{attribute 'pack_mode':='1'}
TYPE InitToteRequestParams :
STRUCT
	source_id : ModelIdentifier;
	target_id: ModelIdentifier;
END_STRUCT
END_TYPE

(* stored: Version 1.1.0.1, ProductVersion 3.1.4024.12
   DUT InitToteRequestParams: Id {baeb2183-429b-4331-98cf-72437eb37aec} *)
